// TIA Portal project "CizgiIzleyenRobot" (V17)

(* hardware
DEVICE "S7-1200 station_1"  S7-1200 Station
   slot 0: "Rack_0"  S7-1200 Rack  Rack  V1.0
   slot 1: "PLC_1"  CPU 1214C DC/DC/DC  6ES7 214-1AG40-0XB0  V4.5
*)

// ===== PLC "PLC_1"  CPU 1214C DC/DC/DC =====

VAR_GLOBAL   // PLC tag table "Default tag table"
   "MANUAL / AUTOMATIC SECIM ANAHTARI" AT %I0.4 : Bool;
   "LİMİT SWİTCH 1" AT %I0.0 : Bool;
   "YUKARI START" AT %I0.6 : Bool;
   "Tag_4" AT %M60.0 : Bool;
   "YUKARI OTOMATİK" AT %M10.0 : Bool;
   "ASAGI OTOMATIK" AT %M10.1 : Bool;
   "Tag_2" AT %M60.1 : Bool;
   "LİMİT SWİTCH 2" AT %I0.3 : Bool;
   "ASAGI START" AT %I10.7 : Bool;
   "Tag_1" AT %M60.2 : Bool;
   "Tag_3" AT %M60.3 : Bool;
   "AŞAĞI YÖN" AT %Q0.1 : Bool;
   "Tag_6" AT %M60.4 : Bool;
   "YUKARI YÖN MERKER'İ" AT %M10.5 : Bool;
   "Tag_7" AT %M60.5 : Bool;
   "YUKARI YÖN" AT %Q0.0 : Bool;
   "YUKARI MANUAL" AT %M10.2 : Bool;
   "YUKARI START(1)" AT %I10.6 : Bool;
   "AŞAĞI START" AT %I0.7 : Bool;
   "AŞAĞI MANUAL" AT %M10.3 : Bool;
   "Tag_5" AT %M60.6 : Bool;
   "AŞAĞI YÖN MERKERİ" AT %M10.4 : Bool;
   "Tag_8" AT %M60.7 : Bool;
   "Tag_9" AT %M70.0 : Bool;
   "YAVAŞLATMA SWİTCH -1" AT %I0.1 : Bool;
   "YAVAŞLATMA SWİTCH -2" AT %I0.2 : Bool;
   "Tag_10" AT %M70.1 : Bool;
   "HIZ-1 MERKERİ" AT %M10.6 : Bool;
   "YÜKSEK DEVİR ÇALIŞMA 1.ÇIKIŞ" AT %Q0.3 : Bool;
   "DÜŞÜK DEVİR ÇIKIŞI" AT %Q0.2 : Bool;
   "Tag_11" AT %M70.2 : Bool;
   "Tag_12" AT %M70.3 : Bool;
   "HIZ-2 MERKERİ" AT %M10.7 : Bool;
   "YÜKSEK DEVİR ÇALIŞMA 2.ÇIKIŞ" AT %Q0.4 : Bool;
END_VAR

ORGANIZATION_BLOCK "Main"   // OB1, LAD, ProgramCycle
TITLE = "Main Program Sweep (Cycle)"
{ S7_Optimized_Access := 'TRUE' }
VERSION : 0.1
   VAR_INPUT
      Initial_Call : Bool;   // Initial call of this OB
      Remanence : Bool;   // =True, if remanent data are available
   END_VAR
   VAR_TEMP   // added for the SCL form of the ladder/FBD networks
      _w1 : Bool;
      _w2 : Bool;
      _w3 : Bool;
      _w4 : Bool;
   END_VAR
BEGIN

REGION Network 1
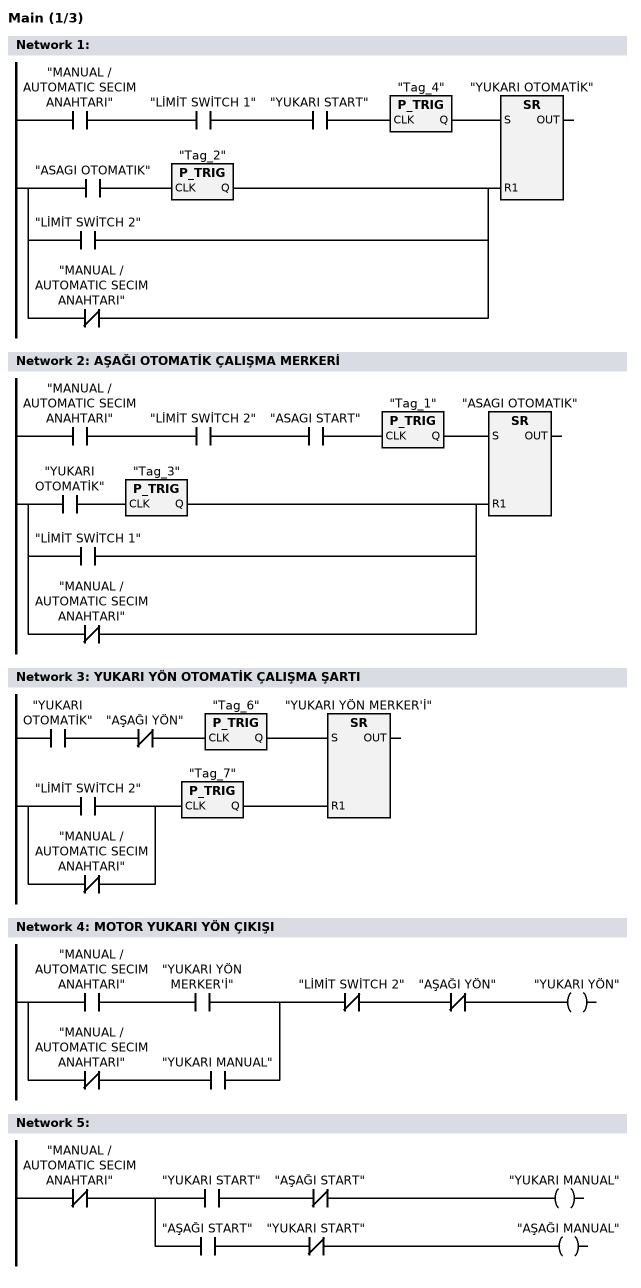
   RUNG wire#powerrail
      Contact( "MANUAL / AUTOMATIC SECIM ANAHTARI" )
      Contact( "LİMİT SWİTCH 1" )
      Contact( "YUKARI START" )
      P_Trig( "Tag_4" )
      S_SR(operand := "YUKARI OTOMATİK", r1 := wire#w1)
   END_RUNG
   RUNG wire#powerrail
      Contact( "ASAGI OTOMATIK" )
      P_Trig( "Tag_2" )
   END_RUNG wire#w1
   RUNG wire#powerrail
      Contact( "LİMİT SWİTCH 2" )
   END_RUNG wire#w1
   RUNG wire#powerrail
      I_Contact( "MANUAL / AUTOMATIC SECIM ANAHTARI" )
   END_RUNG wire#w1
   // the same network as SCL:
   #_w1 := "MANUAL / AUTOMATIC SECIM ANAHTARI" AND "LİMİT SWİTCH 1" AND "YUKARI START";
   #_w2 := #_w1 AND NOT "Tag_4";   // rising edge
   "Tag_4" := #_w1;
   #_w3 := "ASAGI OTOMATIK" AND NOT "Tag_2";   // rising edge
   "Tag_2" := "ASAGI OTOMATIK";
   IF #_w2 THEN
       "YUKARI OTOMATİK" := TRUE;   // SR flip-flop
   END_IF;
   IF #_w3 OR "LİMİT SWİTCH 2" OR NOT "MANUAL / AUTOMATIC SECIM ANAHTARI" THEN
       "YUKARI OTOMATİK" := FALSE;
   END_IF;
END_REGION

REGION Network 2: AŞAĞI OTOMATİK ÇALIŞMA MERKERİ
   RUNG wire#powerrail
      Contact( "MANUAL / AUTOMATIC SECIM ANAHTARI" )
      Contact( "LİMİT SWİTCH 2" )
      Contact( "ASAGI START" )
      P_Trig( "Tag_1" )
      S_SR(operand := "ASAGI OTOMATIK", r1 := wire#w1)
   END_RUNG
   RUNG wire#powerrail
      Contact( "YUKARI OTOMATİK" )
      P_Trig( "Tag_3" )
   END_RUNG wire#w1
   RUNG wire#powerrail
      Contact( "LİMİT SWİTCH 1" )
   END_RUNG wire#w1
   RUNG wire#powerrail
      I_Contact( "MANUAL / AUTOMATIC SECIM ANAHTARI" )
   END_RUNG wire#w1
   // the same network as SCL:
   #_w1 := "MANUAL / AUTOMATIC SECIM ANAHTARI" AND "LİMİT SWİTCH 2" AND "ASAGI START";
   #_w2 := #_w1 AND NOT "Tag_1";   // rising edge
   "Tag_1" := #_w1;
   #_w3 := "YUKARI OTOMATİK" AND NOT "Tag_3";   // rising edge
   "Tag_3" := "YUKARI OTOMATİK";
   IF #_w2 THEN
       "ASAGI OTOMATIK" := TRUE;   // SR flip-flop
   END_IF;
   IF #_w3 OR "LİMİT SWİTCH 1" OR NOT "MANUAL / AUTOMATIC SECIM ANAHTARI" THEN
       "ASAGI OTOMATIK" := FALSE;
   END_IF;
END_REGION

REGION Network 3: YUKARI YÖN OTOMATİK ÇALIŞMA ŞARTI
   RUNG wire#powerrail
      Contact( "YUKARI OTOMATİK" )
      I_Contact( "AŞAĞI YÖN" )
      P_Trig( "Tag_6" )
      S_SR(operand := "YUKARI YÖN MERKER'İ", r1 := wire#w2)
   END_RUNG
   RUNG wire#powerrail
      Contact( "LİMİT SWİTCH 2" )
      wire#w1
      P_Trig( "Tag_7" )
   END_RUNG wire#w2
   RUNG wire#powerrail
      I_Contact( "MANUAL / AUTOMATIC SECIM ANAHTARI" )
   END_RUNG wire#w1
   // the same network as SCL:
   #_w1 := "YUKARI OTOMATİK" AND NOT "AŞAĞI YÖN";
   #_w2 := #_w1 AND NOT "Tag_6";   // rising edge
   "Tag_6" := #_w1;
   #_w3 := "LİMİT SWİTCH 2" OR NOT "MANUAL / AUTOMATIC SECIM ANAHTARI";
   #_w4 := #_w3 AND NOT "Tag_7";   // rising edge
   "Tag_7" := #_w3;
   IF #_w2 THEN
       "YUKARI YÖN MERKER'İ" := TRUE;   // SR flip-flop
   END_IF;
   IF #_w4 THEN "YUKARI YÖN MERKER'İ" := FALSE; END_IF;
END_REGION

REGION Network 4: MOTOR YUKARI YÖN ÇIKIŞI
   RUNG wire#powerrail
      Contact( "MANUAL / AUTOMATIC SECIM ANAHTARI" )
      Contact( "YUKARI YÖN MERKER'İ" )
      wire#w1
      I_Contact( "LİMİT SWİTCH 2" )
      I_Contact( "AŞAĞI YÖN" )
      Coil( "YUKARI YÖN" )
   END_RUNG
   RUNG wire#powerrail
      I_Contact( "MANUAL / AUTOMATIC SECIM ANAHTARI" )
      Contact( "YUKARI MANUAL" )
   END_RUNG wire#w1
   // the same network as SCL:
   "YUKARI YÖN" := (("MANUAL / AUTOMATIC SECIM ANAHTARI" AND "YUKARI YÖN MERKER'İ") OR (NOT "MANUAL / AUTOMATIC SECIM ANAHTARI" AND "YUKARI MANUAL")) AND NOT "LİMİT SWİTCH 2" AND NOT "AŞAĞI YÖN";
END_REGION

REGION Network 5
   RUNG wire#powerrail
      I_Contact( "MANUAL / AUTOMATIC SECIM ANAHTARI" )
      wire#w1
      Contact( "YUKARI START" )
      I_Contact( "AŞAĞI START" )
      Coil( "YUKARI MANUAL" )
   END_RUNG
   RUNG wire#w1
      Contact( "AŞAĞI START" )
      I_Contact( "YUKARI START" )
      Coil( "AŞAĞI MANUAL" )
   END_RUNG
   // the same network as SCL:
   #_w1 := NOT "MANUAL / AUTOMATIC SECIM ANAHTARI";
   "YUKARI MANUAL" := #_w1 AND "YUKARI START" AND NOT "AŞAĞI START";
   "AŞAĞI MANUAL" := #_w1 AND "AŞAĞI START" AND NOT "YUKARI START";
END_REGION

REGION Network 6
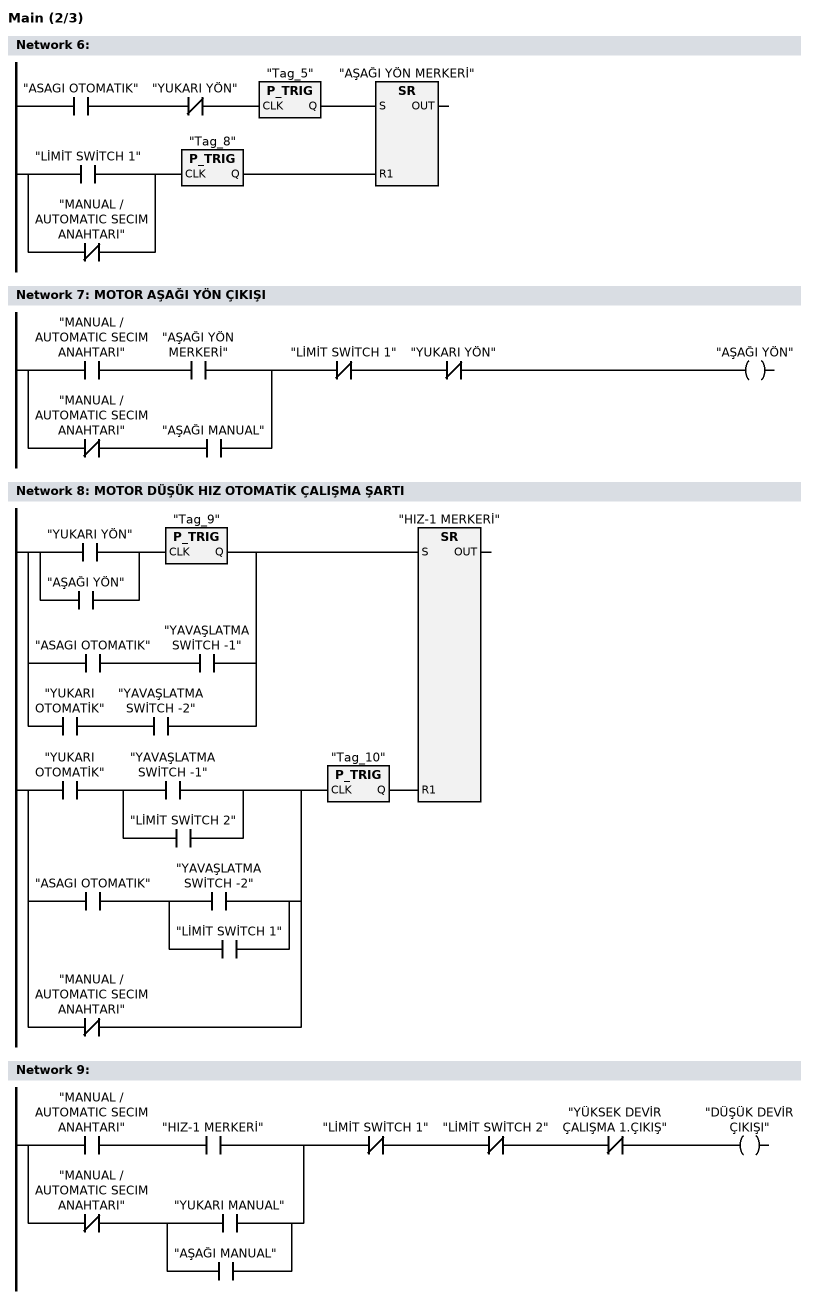
   RUNG wire#powerrail
      Contact( "ASAGI OTOMATIK" )
      I_Contact( "YUKARI YÖN" )
      P_Trig( "Tag_5" )
      S_SR(operand := "AŞAĞI YÖN MERKERİ", r1 := wire#w2)
   END_RUNG
   RUNG wire#powerrail
      Contact( "LİMİT SWİTCH 1" )
      wire#w1
      P_Trig( "Tag_8" )
   END_RUNG wire#w2
   RUNG wire#powerrail
      I_Contact( "MANUAL / AUTOMATIC SECIM ANAHTARI" )
   END_RUNG wire#w1
   // the same network as SCL:
   #_w1 := "ASAGI OTOMATIK" AND NOT "YUKARI YÖN";
   #_w2 := #_w1 AND NOT "Tag_5";   // rising edge
   "Tag_5" := #_w1;
   #_w3 := "LİMİT SWİTCH 1" OR NOT "MANUAL / AUTOMATIC SECIM ANAHTARI";
   #_w4 := #_w3 AND NOT "Tag_8";   // rising edge
   "Tag_8" := #_w3;
   IF #_w2 THEN
       "AŞAĞI YÖN MERKERİ" := TRUE;   // SR flip-flop
   END_IF;
   IF #_w4 THEN "AŞAĞI YÖN MERKERİ" := FALSE; END_IF;
END_REGION

REGION Network 7: MOTOR AŞAĞI YÖN ÇIKIŞI
   RUNG wire#powerrail
      Contact( "MANUAL / AUTOMATIC SECIM ANAHTARI" )
      Contact( "AŞAĞI YÖN MERKERİ" )
      wire#w1
      I_Contact( "LİMİT SWİTCH 1" )
      I_Contact( "YUKARI YÖN" )
      Coil( "AŞAĞI YÖN" )
   END_RUNG
   RUNG wire#powerrail
      I_Contact( "MANUAL / AUTOMATIC SECIM ANAHTARI" )
      Contact( "AŞAĞI MANUAL" )
   END_RUNG wire#w1
   // the same network as SCL:
   "AŞAĞI YÖN" := (("MANUAL / AUTOMATIC SECIM ANAHTARI" AND "AŞAĞI YÖN MERKERİ") OR (NOT "MANUAL / AUTOMATIC SECIM ANAHTARI" AND "AŞAĞI MANUAL")) AND NOT "LİMİT SWİTCH 1" AND NOT "YUKARI YÖN";
END_REGION

REGION Network 8: MOTOR DÜŞÜK HIZ OTOMATİK ÇALIŞMA ŞARTI
   RUNG wire#powerrail
      Contact( "YUKARI YÖN" )
      wire#w1
      P_Trig( "Tag_9" )
      wire#w2
      S_SR(operand := "HIZ-1 MERKERİ", r1 := wire#w6)
   END_RUNG
   RUNG wire#powerrail
      Contact( "AŞAĞI YÖN" )
   END_RUNG wire#w1
   RUNG wire#powerrail
      Contact( "ASAGI OTOMATIK" )
      Contact( "YAVAŞLATMA SWİTCH -1" )
   END_RUNG wire#w2
   RUNG wire#powerrail
      Contact( "YUKARI OTOMATİK" )
      Contact( "YAVAŞLATMA SWİTCH -2" )
   END_RUNG wire#w2
   RUNG wire#powerrail
      Contact( "YUKARI OTOMATİK" )
      wire#w3
      Contact( "YAVAŞLATMA SWİTCH -1" )
      wire#w4
      P_Trig( "Tag_10" )
   END_RUNG wire#w6
   RUNG wire#w3
      Contact( "LİMİT SWİTCH 2" )
   END_RUNG wire#w4
   RUNG wire#powerrail
      Contact( "ASAGI OTOMATIK" )
      wire#w5
      Contact( "YAVAŞLATMA SWİTCH -2" )
   END_RUNG wire#w4
   RUNG wire#w5
      Contact( "LİMİT SWİTCH 1" )
   END_RUNG wire#w4
   RUNG wire#powerrail
      I_Contact( "MANUAL / AUTOMATIC SECIM ANAHTARI" )
   END_RUNG wire#w4
   // the same network as SCL:
   #_w1 := "YUKARI YÖN" OR "AŞAĞI YÖN";
   #_w2 := #_w1 AND NOT "Tag_9";   // rising edge
   "Tag_9" := #_w1;
   #_w3 := ("YUKARI OTOMATİK" AND ("YAVAŞLATMA SWİTCH -1" OR "LİMİT SWİTCH 2")) OR ("ASAGI OTOMATIK" AND ("YAVAŞLATMA SWİTCH -2" OR "LİMİT SWİTCH 1")) OR NOT "MANUAL / AUTOMATIC SECIM ANAHTARI";
   #_w4 := #_w3 AND NOT "Tag_10";   // rising edge
   "Tag_10" := #_w3;
   IF #_w2 OR ("ASAGI OTOMATIK" AND "YAVAŞLATMA SWİTCH -1") OR ("YUKARI OTOMATİK" AND "YAVAŞLATMA SWİTCH -2") THEN
       "HIZ-1 MERKERİ" := TRUE;   // SR flip-flop
   END_IF;
   IF #_w4 THEN "HIZ-1 MERKERİ" := FALSE; END_IF;
END_REGION

REGION Network 9
   RUNG wire#powerrail
      Contact( "MANUAL / AUTOMATIC SECIM ANAHTARI" )
      Contact( "HIZ-1 MERKERİ" )
      wire#w1
      I_Contact( "LİMİT SWİTCH 1" )
      I_Contact( "LİMİT SWİTCH 2" )
      I_Contact( "YÜKSEK DEVİR ÇALIŞMA 1.ÇIKIŞ" )
      Coil( "DÜŞÜK DEVİR ÇIKIŞI" )
   END_RUNG
   RUNG wire#powerrail
      I_Contact( "MANUAL / AUTOMATIC SECIM ANAHTARI" )
      wire#w2
      Contact( "YUKARI MANUAL" )
   END_RUNG wire#w1
   RUNG wire#w2
      Contact( "AŞAĞI MANUAL" )
   END_RUNG wire#w1
   // the same network as SCL:
   "DÜŞÜK DEVİR ÇIKIŞI" := (("MANUAL / AUTOMATIC SECIM ANAHTARI" AND "HIZ-1 MERKERİ") OR (NOT "MANUAL / AUTOMATIC SECIM ANAHTARI" AND ("YUKARI MANUAL" OR "AŞAĞI MANUAL"))) AND NOT "LİMİT SWİTCH 1" AND NOT "LİMİT SWİTCH 2" AND NOT "YÜKSEK DEVİR ÇALIŞMA 1.ÇIKIŞ";
END_REGION

REGION Network 10: MOTOR YÜKSEK HIZ OTOMATİK ÇALIŞMA ŞARTI
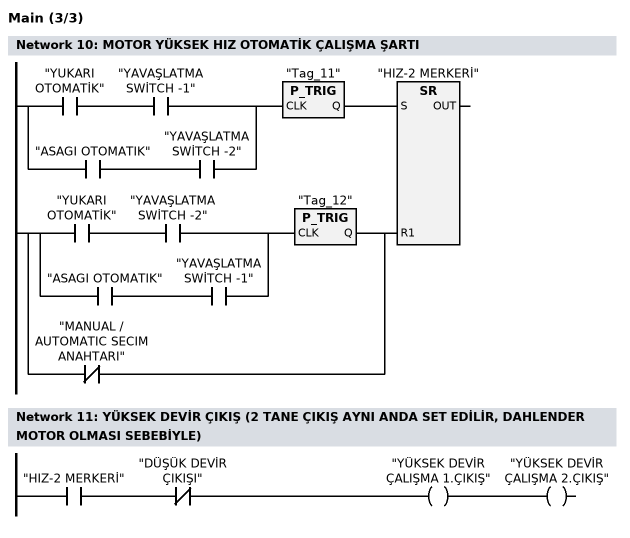
   RUNG wire#powerrail
      Contact( "YUKARI OTOMATİK" )
      Contact( "YAVAŞLATMA SWİTCH -1" )
      wire#w1
      P_Trig( "Tag_11" )
      S_SR(operand := "HIZ-2 MERKERİ", r1 := wire#w3)
   END_RUNG
   RUNG wire#powerrail
      Contact( "ASAGI OTOMATIK" )
      Contact( "YAVAŞLATMA SWİTCH -2" )
   END_RUNG wire#w1
   RUNG wire#powerrail
      Contact( "YUKARI OTOMATİK" )
      Contact( "YAVAŞLATMA SWİTCH -2" )
      wire#w2
      P_Trig( "Tag_12" )
   END_RUNG wire#w3
   RUNG wire#powerrail
      Contact( "ASAGI OTOMATIK" )
      Contact( "YAVAŞLATMA SWİTCH -1" )
   END_RUNG wire#w2
   RUNG wire#powerrail
      I_Contact( "MANUAL / AUTOMATIC SECIM ANAHTARI" )
   END_RUNG wire#w3
   // the same network as SCL:
   #_w1 := ("YUKARI OTOMATİK" AND "YAVAŞLATMA SWİTCH -1") OR ("ASAGI OTOMATIK" AND "YAVAŞLATMA SWİTCH -2");
   #_w2 := #_w1 AND NOT "Tag_11";   // rising edge
   "Tag_11" := #_w1;
   #_w3 := ("YUKARI OTOMATİK" AND "YAVAŞLATMA SWİTCH -2") OR ("ASAGI OTOMATIK" AND "YAVAŞLATMA SWİTCH -1");
   #_w4 := #_w3 AND NOT "Tag_12";   // rising edge
   "Tag_12" := #_w3;
   IF #_w2 THEN
       "HIZ-2 MERKERİ" := TRUE;   // SR flip-flop
   END_IF;
   IF #_w4 OR NOT "MANUAL / AUTOMATIC SECIM ANAHTARI" THEN "HIZ-2 MERKERİ" := FALSE; END_IF;
END_REGION

REGION Network 11: YÜKSEK DEVİR ÇIKIŞ (2 TANE ÇIKIŞ AYNI ANDA SET EDİLİR, DAHLENDER MOTOR OLMASI SEBEBİYLE)
   RUNG wire#powerrail
      Contact( "HIZ-2 MERKERİ" )
      I_Contact( "DÜŞÜK DEVİR ÇIKIŞI" )
      Coil( "YÜKSEK DEVİR ÇALIŞMA 1.ÇIKIŞ" )
      Coil( "YÜKSEK DEVİR ÇALIŞMA 2.ÇIKIŞ" )
   END_RUNG
   // the same network as SCL:
   "YÜKSEK DEVİR ÇALIŞMA 1.ÇIKIŞ" := "HIZ-2 MERKERİ" AND NOT "DÜŞÜK DEVİR ÇIKIŞI";
   "YÜKSEK DEVİR ÇALIŞMA 2.ÇIKIŞ" := "YÜKSEK DEVİR ÇALIŞMA 1.ÇIKIŞ";
END_REGION
END_ORGANIZATION_BLOCK